# B&R Automation Studio project TD52 (part 10)

```c
/******************************************************************************
 * END OF CODE
 ******************************************************************************/
/*
Local Variables:
c-file-style: bsd
c-basic-offset: 2
comment-column: 45
End:
 */
```

#### MBTMaster.h
```c
/*****************************************************************************
 * Copyright:    B&R Industrie-Automation AG
 *
 * Project:      Library MBTCP
 *
 * Target:       B&R-PCC
 *
 * AR-Version:   B 2.01
 *
 * AS-Version:   V 3.0.71.16.SP01
 *
 * Filename:     MBTMaster.h
 *
 * Function:     module-description
 *
 * Dependencies: description of all dependencies
 *
 *****************************************************************************
 * History:
 *
 * Version | Date        | Author      | Description
 * --------------------------------------------------------------------------
 *    1.00 | 2008-Sep-30 | H.Anderes    | creation
 *****************************************************************************/

/*****************************************************************************
 * includes
 *****************************************************************************/
#ifndef MBTMASTER_H_
#define MBTMASTER_H_
/* ansi-c import */
#include <string.h>
/* system import */
#include <bur/plc.h>                         /* IEC data types */
#include <asstring.h>
#include <brsystem.h>
#include <astcp.h>
#include <convert.h>
#include <sys_lib.h>
/* user defined import */
#include "MBTCP.h"

/*#define _MBTCP_LOGGER_DEBUG*/    /* if defined, errors are logged into the logger */
/*#define _MBTCP_LOGGER_EVENT*/    /* if defined, events are logged into the logger */

#ifdef __i386__
#define SWAPUINT        swapUINT
#define SWAPINT         swapINT
#else
#define SWAPUINT
#define SWAPINT
#endif

/*****************************************************************************
 * constants / macros
 *****************************************************************************/
#define NELEMS(array)           (sizeof(array) / sizeof(array[0]))
/* Booleans, switches
 */
enum {
  FALSE                   = 0,
  TRUE                    = 1,
  EXIT_FAILURE            = 1,
  ON                      = 0xFF00,
  OFF                     = 0x0000
};

#define MAX_COILS    2000
#define MAX_REGISTER 127
/*****************************************************************************
 * type definitions
 *****************************************************************************/
/* STEP values
 */
enum {
  INIT                    = 0,
  WAIT_SERVER             = 5,
  OPEN_PORT               = 10,
  IOCTL                   = 15,
  WAIT_CONNECTION         = 20,
  WAIT_REQUEST            = 30,
  SEND_ANSWER             = 40,
  SEND_REQUEST            = 50,
  WAIT_ANSWER             = 60,
  CLOSE_PORT              = 70,
  FATAL_ERROR0            = 240,
  FATAL_ERROR1            = 241,
  FATAL_ERROR2            = 242,
  FATAL_ERROR3            = 243,
  FATAL_ERROR4            = 244,
  FATAL_ERROR5            = 245,
  FATAL_ERROR6            = 246,
  FATAL_ERROR7            = 247,
  FATAL_ERROR8            = 248,
  FATAL_ERROR9            = 249,
  FATAL_ERROR10           = 250,
  FATAL_ERROR             = 251,
  FINAL_ERROR			  = 252,

  DISABLE                 = 65534,
  BUSY                    = 65535
};

/* Modbus function codes
 */
enum {
  READ_COILS                            = 0x01,
  READ_DISCRETE_INPUTS                  = 0x02,
  READ_HOLDING_REGISTERS                = 0x03,
  READ_INPUT_REGISTERS                  = 0x04,
  WRITE_SINGLE_COIL                     = 0x05,
  WRITE_SINGLE_REGISTER                 = 0x06,
  WRITE_MULTIPLE_COILS                  = 0x0F,
  WRITE_MULTIPLE_REGISTERS              = 0x10,
  READ_WRITE_MULTIPLE_REGISTERS         = 0x17
};
/* Modbus protocol exception codes
 */
enum {
  MB_ILLEGAL_FUNCTION                   = 0x01,
  MB_ILLEGAL_DATA_ADDRESS               = 0x02,
  MB_ILLEGAL_DATA_VALUE                 = 0x03,
  MB_SLAVE_DEVICE_FAILURE               = 0x04,
  MB_ACKNOWLEDGE                        = 0x05,
  MB_SLAVE_DEVICE_BUSY                  = 0x06,
  MB_MEMORY_PARITY_ERROR                = 0x08,
  MB_GATEWAY_PATH_UNAVAILABLE           = 0x0A,
  MB_GATEWAY_TARGET_DEV_FAILED_RESPOND  = 0x0B
};
/* Dimensions
 */
enum {
  MBT_SLAVE_PORT        = 502,
  MAX_OPEN_RETRIES      = 3,
  RECV_TIMEOUT_DFLT     = 500,               /* default timeout */
  IPADDR_L              = 18,
  MAX_NBR_REQUESTS      = 5,                 /* was 20 */
  MAX_BUFFER_LEN        = 1200,/*128,*/
  MESS_LEN              = 100,               /* error message length */
};

/* Datatypes */
typedef struct MBTMasterActionParam_typ
{
  USINT usiFCode;
  USINT usiUnit;
  UINT  uiReadAddr;
  UINT  uiReadQty;
  UDINT puiReadVal;
  UINT  uiWriteAddr;
  UINT  uiWriteQty;
  UDINT puiWriteVal;
  UDINT udiTimer;
} MBTMasterActionParam_typ;

typedef struct MBTMasterActionEnable_typ
{
  BOOL bCyclic;
  BOOL bSingle;
} MBTMasterActionEnable_typ;

typedef struct tstMBT_MData
{
  MBTMasterActionEnable_typ actEnable[MAX_NBR_REQUESTS];
  MBTMasterActionParam_typ actParam[MAX_NBR_REQUESTS];
} tstMBT_MData;

typedef struct
{
  BOOL                  bEnable;
  STRING                slvIPAddr[IPADDR_L];
  UINT                  uiPort;
  UINT                  uiRecvTimeout;
  UDINT                 udiCycleTime;
  tstMBT_MData*         pData;
  UINT                  uiStep;
  TcpOpen_typ           stTcpOpen;
  TcpIoctl_typ          stTcpIoctl;
  TcpClient_typ         stTcpClient;
  TcpSend_typ           stTcpSend;
  TcpRecv_typ           stTcpRecv;
  TcpClose_typ          stTcpClose;
  USINT                 usiLastReq;
  UDINT                 udiRecvTimer;
  UDINT                 udiSendTimer[MAX_NBR_REQUESTS];
  USINT                 usiSendBuf[MAX_BUFFER_LEN];
  USINT                 usiRecvBuf[MAX_BUFFER_LEN];
  BOOL                  bRecvOK;
  UINT                  uiStatus;
  UINT                  uiTxID;
  UDINT                 udiWrongMsg;
  STRING                szMsg[MESS_LEN];
  tcpLINGER_typ         mLinger;
  USINT                 usiOpenRetries;
  USINT                 usiSendCnt;
} tstMBT_MVars;

/*****************************************************************************
 * functions protoytpes
 ****************************************************************************/
void  fMBTMStates(tstMBT_MVars* inst);
UINT create_request_to_server(tstMBT_MVars*   inst,
                               tstMBT_MData*   config,
                               USINT           usiOp,
                               USINT*          usiSendBuf,
                               UINT            uiTxID);
USINT analyze_answer_from_server(tstMBT_MVars* inst,
                                 tstMBT_MData* config,
                                 USINT         usiOp,
                                 USINT*        usiRecvBuf,
                                 UINT          uiTxID);

/****************************************************************************
 * END OF CODE
 ****************************************************************************/
/*
Local Variables:
c-file-style: bsd
c-basic-offset: 2
comment-column: 45
End:
 */
#endif /* MBTMASTER_H_ */
```

#### MBTMaster.c
```c
/******************************************************************************
 * Copyright:    B&R Industrie-Automation AG
 *
 * Project:      Library MBTCP
 *
 * Target:       B&R-PCC
 *
 * AR-Version:   B 2.01
 *
 * AS-Version:   V 3.0.71.16.SP01
 *
 * Filename:     MBTMaster.c
 *
 * Function:     module-description
 *
 * Dependencies: description of all dependencies
 *
 ******************************************************************************
 * History:
 *
 * Version | Date        | Author      | Description
 * ----------------------------------------------------------------------------
 *    1.00 | 2008-Sep-30 | H.Anderes   | creation
 *    2.00 | 2010-okt-04 | H.Anderes   | refactory
 *    5.00 | 2021-may-07 | W.Froehlich | set correct FUB state fMBTSClose.uiStatus
 *****************************************************************************/

/******************************************************************************
 * includes
 *****************************************************************************/
/* ansi-c import */
/* system import */
/* user defined import */
#include "MBTMaster.h"

/******************************************************************************
 * functions
 ******************************************************************************/
/*============================================================================*/
void fMBTMStates(tstMBT_MVars* inst)
/*----------------------------------------------------------------------------
  Function:

  History:

  Version | Date        | Author      | Description
  ----------------------------------------------------------------------------
  1.00    | 2008-sep-30 | H.Anderes    | creation
  2.00    | 2010-okt-04 | H.Anderes   | refactory
  ============================================================================*/
{
  /* _LOCAL */
  UINT uiFatalErrNum;
  USINT i, usiOp;                            /* usiOp: number of operations */
  USINT recv_status;
  /* _DYNAMIC */
  /*==========================================================================*/
  /* check if a null pointer is passed to the fub */
  if (inst == NULL)
  {
    return;
  }
  /*--------------------------------------------------------------------------------
    state machine : Modbus TCP Master
  ---------------------------------------------------------------------------------*/
  switch(inst->uiStep)
  {
  /*-----------------------------------------------------------------------------
    INIT: initialize TcpSend and TCPRecv
  ------------------------------------------------------------------------------*/
  case INIT:
    inst->stTcpSend.pData   = (UDINT)inst->usiSendBuf;
    inst->stTcpRecv.pData   = (UDINT)inst->usiRecvBuf;
    inst->stTcpRecv.datamax = MAX_BUFFER_LEN;
    inst->uiStep            = DISABLE;
    /* FALL THROUGH */
  /*-----------------------------------------------------------------------------
    DISBALE: waits until the fub is enabled
  ------------------------------------------------------------------------------*/
  case DISABLE:
    if(inst->bEnable)
    {
      inst->uiStep = OPEN_PORT;
    }
    break;
  /*-----------------------------------------------------------------------------
    OPEN: opens a TCP - socket
  ------------------------------------------------------------------------------*/
  case OPEN_PORT:
    inst->stTcpOpen.enable = 1;
    inst->stTcpOpen.port   = 0;
    /* call TcpOpen() */
    TcpOpen(&inst->stTcpOpen);
    /* verfiy status */
    switch (inst->stTcpOpen.status)
    {
    /*-------------------------------------------------------------------------*/
    case ERR_OK:
      inst->stTcpClient.enable     = 1;
      inst->stTcpClient.ident      = inst->stTcpOpen.ident;
      inst->stTcpClient.pServer    = (UDINT)inst->slvIPAddr;
      inst->stTcpClient.portserv   = inst->uiPort;
      inst->stTcpSend.ident        = inst->stTcpOpen.ident;
      inst->stTcpRecv.ident        = inst->stTcpOpen.ident;
      inst->uiStep                 = IOCTL;
      /************************************************************************/
      #ifdef _MBTCP_LOGGER_EVENT
	     ERRxwarning( mbtEVENT_OPEN_PORT,
                   inst->stTcpOpen.ident,
                   "MBTCP Client: Open Port");
      #endif
      /************************************************************************/
      break;
    /*-------------------------------------------------------------------------*/
    case ERR_FUB_BUSY:
      /* do nothing */
      break;
    /*-------------------------------------------------------------------------*/
    case tcpERR_NOMORE_IDENTS:
    case tcpERR_ALREADY_EXIST:
    case tcpERR_SOCKET_CREATE:
    case tcpERR_SOCKET_BIND:
    case tcpERR_INTERFACE:
    case tcpERR_SYSTEM:
    case ERR_FUB_ENABLE_FALSE:
    default:
      inst->uiStatus = inst->stTcpOpen.status;
      inst->uiStep   = FATAL_ERROR0;
      break;
    }
    break;
  /*-----------------------------------------------------------------------------
    IOCTRL: configuration of the TCP - connection
  ------------------------------------------------------------------------------*/
  case IOCTL:
    /* set linger that the connection is not abort immediately */
    inst->mLinger.lOnOff     = 0;
    inst->mLinger.lLinger    = 0;
     /* initialize fub */
    inst->stTcpIoctl.enable 	= 1;
    inst->stTcpIoctl.ident	  = inst->stTcpOpen.ident;
    inst->stTcpIoctl.ioctl 	 = tcpSO_LINGER_SET;
    inst->stTcpIoctl.pData	  = (UDINT)&inst->mLinger;
    inst->stTcpIoctl.datalen	= sizeof(tcpLINGER_typ);
    /* call  TcpIoctl()n */
    TcpIoctl(&inst->stTcpIoctl);
    /* verify status */
    switch (inst->stTcpIoctl.status)
    {
    /*-------------------------------------------------------------------------*/
    case ERR_OK:
      inst->usiOpenRetries = 0;      /* we reset prior to next step */
      inst->uiStep         = WAIT_CONNECTION;
      break;
    /*-------------------------------------------------------------------------*/
    case ERR_FUB_BUSY:
      inst->uiStep = IOCTL;
      break;
    /*-------------------------------------------------------------------------*/
    case tcpERR_INVALID_IDENT:
      inst->uiStatus = inst->stTcpIoctl.status;
      if (inst->usiOpenRetries < MAX_OPEN_RETRIES)
      {
        inst->uiStep = OPEN_PORT;
        inst->usiOpenRetries++;
        /************************************************************************/
        #ifdef _MBTCP_LOGGER_DEBUG
		      ERRxwarning( mbtERR_OPEN_RETRIES_IOC,
                     inst->stTcpOpen.ident,
                     "MBTCP Client: OPEN Retries IOCTL");
        #endif
        /************************************************************************/
      }
      else
      {
        inst->uiStep = FATAL_ERROR1;
      }
      break;
    /*-------------------------------------------------------------------------*/
    case tcpERR_PARAMETER:
      inst->uiStatus = inst->stTcpIoctl.status;
      inst->uiStep   = CLOSE_PORT;
      break;
    /*-------------------------------------------------------------------------*/
    case tcpERR_INVALID_IOCTL:
    case ERR_FUB_ENABLE_FALSE:
    default:
      inst->uiStatus = inst->stTcpIoctl.status;
      inst->uiStep   = FATAL_ERROR2;
      break;
    }
    break;
  /*-----------------------------------------------------------------------------
    WAIT: waits until a connection to a TCP Server is acc
  ------------------------------------------------------------------------------*/
  case WAIT_CONNECTION:
    inst->stTcpClient.enable = 1;
    /* call TcpClient() */
    TcpClient(&inst->stTcpClient);
    /* verify status */
    switch (inst->stTcpClient.status)
    {
    /*-------------------------------------------------------------------------*/
    case ERR_OK:
      inst->uiStep = SEND_REQUEST;
      break;
    /*-------------------------------------------------------------------------*/
    case ERR_FUB_BUSY:
      /* do nothing */
	     strcpy( inst->szMsg,
              "WAIT_CONNECTION:TcpClient: Wait Connection");
      break;
    /*-------------------------------------------------------------------------*/
    case tcpERR_INVALID:
   	  inst->uiStep = CLOSE_PORT;
      /*************************************************************************/
      #ifdef _MBTCP_LOGGER_DEBUG
   	  ERRxwarning( tcpERR_INVALID,
                   inst->stTcpClient.ident,
                   "MBTCP Client: Wait connecction; Invalid ");
      #endif
      /*************************************************************************/
      break;
    /*-------------------------------------------------------------------------*/
    case tcpERR_ALREADY_CONNECTED:
      inst->uiStep = CLOSE_PORT;
      /*************************************************************************/
      #ifdef _MBTCP_LOGGER_DEBUG
	     ERRxwarning( tcpERR_ALREADY_CONNECTED,
                             inst->stTcpClient.ident,
                             "MBTCP Client: Wait connecction; Already connected");
      #endif
      /*************************************************************************/
      break;
    /*-------------------------------------------------------------------------*/
    case tcpERR_SYSTEM:
    case ERR_FUB_ENABLE_FALSE:
    default:
      inst->uiStep = FATAL_ERROR3;
      break;
    }
    break;
  /*-----------------------------------------------------------------------------
    CREATE: creates the request
  ------------------------------------------------------------------------------*/
  case SEND_REQUEST:
    if (inst->bEnable)
    {
      inst->bRecvOK = FALSE;
      /* cycle through list of Modbus operations for MAX_NBR_REQUESTS times */
      for (i = inst->usiLastReq + 1;
           i < (MAX_NBR_REQUESTS + inst->usiLastReq + 1);
           i++)
      {
        usiOp = i % MAX_NBR_REQUESTS;
        if ((*(inst->pData)).actEnable[usiOp].bSingle)
        {
          inst->udiSendTimer[usiOp] =
            (*(inst->pData)).actParam[usiOp].udiTimer;
        }
        if ( (((*(inst->pData)).actEnable[usiOp].bCyclic)
              || ((*(inst->pData)).actEnable[usiOp].bSingle)))
        {
          if (inst->udiSendTimer[usiOp]
              >= (*(inst->pData)).actParam[usiOp].udiTimer)
          {
            inst->usiLastReq = usiOp;
            inst->uiStep = SEND_REQUEST + 1;
            inst->uiTxID++;
            inst->stTcpSend.datalen =
                create_request_to_server((tstMBT_MVars*)(inst),
                                       (tstMBT_MData*)(inst->pData),
                                       usiOp,
                                       inst->usiSendBuf,
                                       inst->uiTxID);
            inst->udiSendTimer[usiOp] = 0;
            break;
          }
          else
          {
            inst->udiSendTimer[usiOp] += inst->udiCycleTime;
          }
        }
        else
        {
          inst->udiSendTimer[usiOp]
            = (*(inst->pData)).actParam[usiOp].udiTimer;
        }
      }
    }
    else
    {
      inst->uiStep = CLOSE_PORT;
    }
    break;
  /*-----------------------------------------------------------------------------
    SEND: sends the created request to the server/slave
  ------------------------------------------------------------------------------*/
  case SEND_REQUEST + 1:
    if (inst->bEnable)
    {
      inst->stTcpSend.enable = 1;
      /* call TcpSend() */
      TcpSend(&inst->stTcpSend);
      /* verfiy status */
      switch (inst->stTcpSend.status)
      {
      /*-------------------------------------------------------------------------*/
      case ERR_OK:
        inst->usiSendCnt   = 0;
        inst->udiRecvTimer = 0;
        inst->uiStep       = WAIT_ANSWER;
        break;
      /*-------------------------------------------------------------------------*/
      case ERR_FUB_BUSY:
	       /* do nothing */
		      strcpy( inst->szMsg,
                "SEND_REQUEST + 1:TcpSend: ERR_FUB_BUSY");
	  	    break;
      /*-------------------------------------------------------------------------*/
      case tcpERR_WOULDBLOCK:
         /* send again */
         /************************************************************************/
         #ifdef _MBTCP_LOGGER_DEBUG
  	      ERRxwarning( tcpERR_WOULDBLOCK,
                      inst->stTcpClient.ident,
                      "MBTCP Client: Wouldblock");
         #endif
         /***********************************************************************/
   	   	break;
      /*-------------------------------------------------------------------------*/
      case tcpERR_SENTLEN:
        /* send length not ok. send again */
        /************************************************************************/
        #ifdef _MBTCP_LOGGER_DEBUG
        ERRxwarning( tcpERR_SENTLEN,
                     inst->stTcpClient.ident,
                     "MBTCP Client: Send lenght not Ok");
        #endif
        /************************************************************************/
        break;
      /*------------------------------------------------------------------------*/
      case tcpERR_NOT_CONNECTED:
        inst->uiStep = CLOSE_PORT;
        /************************************************************************/
        #ifdef _MBTCP_LOGGER_DEBUG
		      ERRxwarning( tcpERR_NOT_CONNECTED,
                     inst->stTcpClient.ident,
                     "MBTCP Client: Not connected");
        #endif
        /************************************************************************/
        break;
      /*-------------------------------------------------------------------------*/
      case tcpERR_INVALID_IDENT:
      case tcpERR_PARAMETER:
      case tcpERR_SYSTEM:
      default:
        inst->uiStep = FATAL_ERROR4;
        break;
      }
    }
    else
    {
      inst->uiStep = CLOSE_PORT;
    }
    break;
  /*-----------------------------------------------------------------------------
    WAIT: waits until a response is received or a timeout occured
  ------------------------------------------------------------------------------*/
  case WAIT_ANSWER:
    if (inst->bEnable)
    {
      inst->udiRecvTimer += inst->udiCycleTime;
      if (inst->udiRecvTimer >= inst->uiRecvTimeout)
      {
        /* send again after timeout */
        inst->uiStep = SEND_REQUEST;
        /************************************************************************/
        #ifdef _MBTCP_LOGGER_DEBUG
		      ERRxwarning( mbtERR_TIMEOUT,
                     inst->stTcpClient.ident,
                     "MBTCP Client: Receive Timeout");
        #endif
        /************************************************************************/
        break;
      }
      inst->stTcpRecv.enable = 1;
      /* call TcpRecv() */
      TcpRecv(&(inst->stTcpRecv));
      /* verfiy status */
      switch (inst->stTcpRecv.status)
      {
      /*-------------------------------------------------------------------------*/
      case ERR_OK:
        if (inst->stTcpRecv.recvlen > 8)
        {
          recv_status =
            analyze_answer_from_server((tstMBT_MVars*)(inst),
                                       (tstMBT_MData*)(inst->pData),
                                       inst->usiLastReq,
                                       inst->usiRecvBuf,
                                       inst->uiTxID);
        }
        else
        {
          recv_status = 1;
        }
        if(recv_status)
		      {
           inst->udiWrongMsg++;
           /**********************************************************************/
           #ifdef _MBTCP_LOGGER_DEBUG
 		        ERRxwarning( mbtERR_RESPONSE,
                        inst->stTcpRecv.ident,
                        "MBTCP Client: Response not Ok");
           #endif
           /**********************************************************************/

        }
        else
        {
          (*(inst->pData)).actEnable[inst->usiLastReq].bSingle = 0;
        }
        inst->uiStep = SEND_REQUEST;
        break;
      /*-------------------------------------------------------------------------*/
      case ERR_FUB_BUSY:
      case ERR_FUB_ENABLE_FALSE:
      case tcpERR_NO_DATA:
        /* do nothing */
		      strcpy(inst->szMsg, "WAIT_ANSWER:TcpClient: tcpERR_NO_DATA");
        break;
      /*-------------------------------------------------------------------------*/
      case tcpERR_NOT_CONNECTED:
        inst->uiStep = SEND_REQUEST;
		      strcpy(inst->szMsg, "WAIT_ANSWER:TcpClient: tcpERR_NOT_CONNECTED");
        break;
      /*-------------------------------------------------------------------------*/
      case tcpERR_INVALID_IDENT:
      case tcpERR_PARAMETER:
      case tcpERR_INVALID:
      case tcpERR_NO_OOBDATA:
      case tcpERR_SYSTEM:
      default:
        inst->uiStep = FATAL_ERROR5;
        break;
      }
    }
    else
    {
      inst->uiStep = CLOSE_PORT;
    }
    break;
  /*-----------------------------------------------------------------------------
    CLOSE: closes the TCP - Socket
  ------------------------------------------------------------------------------*/
  case CLOSE_PORT:
    inst->stTcpClose.enable = 1;
    inst->stTcpClose.ident  = inst->stTcpOpen.ident;
    /*
      inst->stTcpClose.how    = tcpSHUT_RD | tcpSHUT_WR;
    */
    inst->stTcpClose.how    = 0;
    /* call TcpClose() */
    TcpClose(&inst->stTcpClose);
    /* verfiy status */
    switch (inst->stTcpClose.status)
    {
    /*-------------------------------------------------------------------------*/
    case ERR_OK:
      inst->uiStep = DISABLE;
      /*************************************************************************/
      #ifdef _MBTCP_LOGGER_DEBUG
	     ERRxwarning( mbtEVENT_CLOSE_PORT,
                   inst->stTcpClose.ident,
                   "MBTCP Client: Close Port");
      #endif
      /*************************************************************************/
      break;
    /*-------------------------------------------------------------------------*/
    case ERR_FUB_BUSY:
      /* do nothing */
      break;
    /*-------------------------------------------------------------------------*/
    case tcpERR_INVALID_IDENT:
      inst->uiStep = WAIT_CONNECTION;
      break;
    /*-------------------------------------------------------------------------*/
    case ERR_FUB_ENABLE_FALSE:
    default:
      inst->uiStep = FATAL_ERROR6;
      break;
    }
    break;
  /*-----------------------------------------------------------------------------
    FATAL ERROR: a fatal error occured
  ------------------------------------------------------------------------------*/
  case FATAL_ERROR0:
  case FATAL_ERROR1:
  case FATAL_ERROR2:
  case FATAL_ERROR3:
  case FATAL_ERROR4:
  case FATAL_ERROR5:
  case FATAL_ERROR6:
  default:
   /* vefiy in which state the fatal error occured */
  	switch(inst->uiStep)
	  {
	  case FATAL_ERROR0: uiFatalErrNum = 0; break;
  	case FATAL_ERROR1: uiFatalErrNum = 1; break;
  	case FATAL_ERROR2: uiFatalErrNum = 2; break;
  	case FATAL_ERROR3: uiFatalErrNum = 3; break;
  	case FATAL_ERROR4: uiFatalErrNum = 4; break;
  	case FATAL_ERROR5: uiFatalErrNum = 5; break;
  	case FATAL_ERROR6: uiFatalErrNum = 6; break;
	  default:
		   uiFatalErrNum = 7; break;
	  }
	   /*************************************************************************/
    #ifdef _MBTCP_LOGGER_DEBUG
   	ERRxwarning( mbtERR_FATAL_ERROR,
                 uiFatalErrNum,
                 "MBTCP Client: FATAL ERROR State Machine");
    #endif
    /*************************************************************************/
   	inst->uiStep = FINAL_ERROR;
    break;

  case FINAL_ERROR:
  	/*Do nothing until Reboot RPS*/
  	break;
  }
}

/*============================================================================*/
UINT create_request_to_server(tstMBT_MVars* inst,
                               tstMBT_MData* config,
                               USINT         usiOp,
                               USINT*        usiSendBuf,
                               UINT          uiTxID)
/*----------------------------------------------------------------------------
  Function:

  History:

  Version | Date        | Author      | Description
  ----------------------------------------------------------------------------
     1.00 | 2008-sep-30 | H.Anderes    | creation
  ============================================================================*/
{
  UINT  uint_var, data_len, i;
  INT  int_var;
  UINT  value;
  UINT  val;
 /*==========================================================================*/
  data_len = 0;

  memset(usiSendBuf, 0, MAX_BUFFER_LEN);
  /* Transaction id: 2 bytes */
  uint_var = SWAPUINT(uiTxID);
  memmove(&usiSendBuf[0], &uint_var, sizeof(uint_var));
  /* Protocol id: 2 bytes */
  uint_var = 0;
  memmove(&usiSendBuf[2], &uint_var, sizeof(uint_var));
  /* Length: 2 bytes */
  /* Unit: 1 byte */
  usiSendBuf[6] = (*config).actParam[usiOp].usiUnit;

  switch((*config).actParam[usiOp].usiFCode)
  {
  /*-------------------------------------------------------------------------
      READ: read coils
  --------------------------------------------------------------------------*/
  case READ_COILS:
    /* Function code: 1 byte */
    usiSendBuf[7] = READ_COILS;
    /* Starting address: 2 bytes */
    uint_var = SWAPUINT((*config).actParam[usiOp].uiReadAddr);
    memmove(&usiSendBuf[8], &uint_var, sizeof(uint_var));
    /* Coils number: 2 bytes */
    uint_var = SWAPUINT((*config).actParam[usiOp].uiReadQty);
    memmove(&usiSendBuf[10], &uint_var, sizeof(uint_var));
    /* Data len */
    data_len = 6;
    inst->bRecvOK = FALSE;
    break;
  /*-------------------------------------------------------------------------
      READ: read discrete inputs
  --------------------------------------------------------------------------*/
  case READ_DISCRETE_INPUTS:
    /* Function code: 1 byte */
    usiSendBuf[7] = READ_DISCRETE_INPUTS;
    /* Starting address: 2 bytes */
    uint_var = SWAPUINT((*config).actParam[usiOp].uiReadAddr);
    memmove(&usiSendBuf[8], &uint_var, sizeof(uint_var));
    /* Inputs number: 2 bytes */
    uint_var = SWAPUINT((*config).actParam[usiOp].uiReadQty);
    memmove(&usiSendBuf[10], &uint_var, sizeof(uint_var));
    /* Data len */
    data_len = 6;
    inst->bRecvOK = FALSE;
    break;
  /*-------------------------------------------------------------------------
      READ: read holding registers
  --------------------------------------------------------------------------*/
  case READ_HOLDING_REGISTERS:
    /* Function code: 1 byte */
    usiSendBuf[7] = READ_HOLDING_REGISTERS;
    /* Starting address: 2 bytes */
    uint_var = SWAPUINT((*config).actParam[usiOp].uiReadAddr);
    memmove(&usiSendBuf[8], &uint_var, sizeof(uint_var));
    /* Holding registers number: 2 bytes */
    uint_var = SWAPUINT((*config).actParam[usiOp].uiReadQty);
    memmove(&usiSendBuf[10], &uint_var, sizeof(uint_var));
    /* Data len */
    data_len = 6;
    inst->bRecvOK = FALSE;
    break;
  /*-------------------------------------------------------------------------
      READ: read input registers
  --------------------------------------------------------------------------*/
  case READ_INPUT_REGISTERS:
    /* Function code: 1 byte */
    usiSendBuf[7] = READ_INPUT_REGISTERS;
    /* Starting address: 2 bytes */
    uint_var = SWAPUINT((*config).actParam[usiOp].uiReadAddr);
    memmove(&usiSendBuf[8], &uint_var, sizeof(uint_var));
    /* Input registers number: 2 bytes */
    uint_var = SWAPUINT((*config).actParam[usiOp].uiReadQty);
    memmove(&usiSendBuf[10], &uint_var, sizeof(uint_var));
    /* Data len */
    data_len = 6;
    inst->bRecvOK = FALSE;
    break;
  /*-------------------------------------------------------------------------
      WRITE: write single coil
  --------------------------------------------------------------------------*/
  case WRITE_SINGLE_COIL:
    /* Function code: 1 byte */
    usiSendBuf[7] = WRITE_SINGLE_COIL;
    /* Starting address: 2 bytes */
    uint_var = SWAPUINT((*config).actParam[usiOp].uiWriteAddr);
    memmove(&usiSendBuf[8], &uint_var, sizeof(uint_var));
    /* Value: 2 bytes */
    memmove(&val, (UINT *)((*config).actParam[usiOp].puiWriteVal), sizeof(UINT));
    if ((BOOL)(val))
      value = ON;
    else
      value = OFF;
    int_var = SWAPUINT(value);
    memmove(&usiSendBuf[10], &int_var, sizeof(int_var));
    /* Data len */
    data_len = 6;
    inst->bRecvOK = FALSE;
    break;
  /*-------------------------------------------------------------------------
      WRITE: write single register
  --------------------------------------------------------------------------*/
  case WRITE_SINGLE_REGISTER:
    /* Function code: 1 byte */
    usiSendBuf[7] = WRITE_SINGLE_REGISTER;
    /* Starting address: 2 bytes */
    uint_var = SWAPUINT((*config).actParam[usiOp].uiWriteAddr);
    memmove(&usiSendBuf[8], &uint_var, sizeof(uint_var));
    /* Value: 2 bytes */
    memmove(&val, (UINT *)(*config).actParam[usiOp].puiWriteVal, sizeof(UINT));
    value = (UINT)(val);
    uint_var = SWAPUINT(value);
    memmove(&usiSendBuf[10], &uint_var, sizeof(uint_var));
    /* Data len */
    data_len = 6;
    inst->bRecvOK = FALSE;
    break;
  /*-------------------------------------------------------------------------
      WRITE: write multiple coils
  --------------------------------------------------------------------------*/
  case WRITE_MULTIPLE_COILS:
    /* Function code: 1 byte */
    usiSendBuf[7] = WRITE_MULTIPLE_COILS;
    /* Starting address: 2 bytes */
    uint_var = SWAPUINT((*config).actParam[usiOp].uiWriteAddr);
    memmove(&usiSendBuf[8], &uint_var, sizeof(uint_var));
    /* Quantity: 2 bytes */
    uint_var = SWAPUINT((*config).actParam[usiOp].uiWriteQty);
    memmove(&usiSendBuf[10], &uint_var, sizeof(uint_var));
    /* Byte count: 1 byte */
    /* Number of usiSendBuf bytes needed to contain data */
    /* less than 8 binary digits: 1 byte */
    if ( (*config).actParam[usiOp].uiWriteQty % 8)
      usiSendBuf[12] = ((*config).actParam[usiOp].uiWriteQty / 8) + 1;
    else      /* more than 8 binary digits: quantity / 8 bytes */
      usiSendBuf[12] = (*config).actParam[usiOp].uiWriteQty / 8;
    /* Coil value: x byte */
    for (i = 0; i < (*config).actParam[usiOp].uiWriteQty; i++)
    {
      memmove(&val,
              (UINT *)((*config).actParam[usiOp].puiWriteVal  +  i * sizeof(UINT)),
              sizeof(UINT));
      if ((BOOL)(val))
        usiSendBuf[13 + (i/8)]
          = usiSendBuf[13 + (i/8)] | (USINT)(0x01 << (i%8));
      else
        usiSendBuf[13 + (i/8)]
          = usiSendBuf[13 + (i/8)] & (USINT)~(0x01 << (i%8));
    }
    /* Data len */
    data_len = 7 + usiSendBuf[12];
    inst->bRecvOK = FALSE;
    break;
  /*-------------------------------------------------------------------------
      WRITE: write multiple registers
  --------------------------------------------------------------------------*/
  case WRITE_MULTIPLE_REGISTERS:
    /* Function code: 1 byte */
    usiSendBuf[7] = WRITE_MULTIPLE_REGISTERS;
    /* Starting address: 2 bytes */
    uint_var = SWAPUINT((*config).actParam[usiOp].uiWriteAddr);
    memmove(&usiSendBuf[8], &uint_var, sizeof(uint_var));
    /* Quantity: 2 bytes */
    uint_var = SWAPUINT((*config).actParam[usiOp].uiWriteQty);
    memmove(&usiSendBuf[10], &uint_var, sizeof(uint_var));
    /* Byte count: 1 byte */
    usiSendBuf[12] = (*config).actParam[usiOp].uiWriteQty * 2;
    /* Coil value: x byte */
    for(i = 0; i < (*config).actParam[usiOp].uiWriteQty; i++)
    {
      value = ((INT*)((*config).actParam[usiOp].puiWriteVal))[i];
      int_var = SWAPINT(value);
      memmove(&usiSendBuf[13 + (i*2)], &int_var, sizeof(int_var));
    }
    /* Data len */
    data_len = 7 + usiSendBuf[12];
    inst->bRecvOK = FALSE;
    break;
  /*-------------------------------------------------------------------------
     READ WRITE:read  write multiple registers
  --------------------------------------------------------------------------*/
  case READ_WRITE_MULTIPLE_REGISTERS:
    /* Function code: 1 byte */
    usiSendBuf[7] = READ_WRITE_MULTIPLE_REGISTERS;
    /* Read starting address: 2 bytes */
    uint_var = SWAPUINT((*config).actParam[usiOp].uiReadAddr);
    memmove(&usiSendBuf[8], &uint_var, sizeof(uint_var));
    /* Read quantity: 2 bytes */
    uint_var = SWAPUINT((*config).actParam[usiOp].uiReadQty);
    memmove(&usiSendBuf[10], &uint_var, sizeof(uint_var));
    /* Write starting address: 2 bytes */
    uint_var = SWAPUINT((*config).actParam[usiOp].uiWriteAddr);
    memmove(&usiSendBuf[12], &uint_var, sizeof(uint_var));
    /* write quantity: 2 bytes */
    uint_var = SWAPUINT((*config).actParam[usiOp].uiWriteQty);
    memmove(&usiSendBuf[14], &uint_var, sizeof(uint_var));
    /* Byte count: 1 byte */
    usiSendBuf[16] = (*config).actParam[usiOp].uiWriteQty * 2;
    /* Coil value: x byte */
    for(i = 0; i < (*config).actParam[usiOp].uiWriteQty; i++)
    {
      value = ((INT*)((*config).actParam[usiOp].puiWriteVal))[i];
      int_var = SWAPINT(value);
      memmove(&usiSendBuf[17 + (i*2)], &int_var, sizeof(int_var));
    }
    /* Data len */
    data_len = 11 + usiSendBuf[16];
    inst->bRecvOK = FALSE;
    break;
  default:
    break;
  }
  /* Length: 2 bytes */
  uint_var = SWAPUINT(data_len);
  memmove(&usiSendBuf[4], &uint_var, sizeof(uint_var));

  return (6 + data_len);
}

 /*==========================================================================*/
USINT analyze_answer_from_server(tstMBT_MVars* inst,
                                 tstMBT_MData* config,
                                 USINT         usiOp,
                                 USINT*        usiRecvBuf,
                                 UINT          uiTxID)
/*----------------------------------------------------------------------------
  Function:

  History:

  Version | Date        | Author      | Description
  ----------------------------------------------------------------------------
     1.00 | 2008-sep-30 | H.Anderes   | creation
     2.00 | 2010-okt-04 | H.Anderes   | refactory
  ============================================================================*/
{
  INT   int_var;
  UINT  uint_var, recv_tr_id, protocol_id, length, uiQty,i;
  USINT unit, function_code;
  UINT  coil_val, di_val;         /* was UDINT */
  /*==========================================================================*/

  coil_val = 0;
  di_val   = 0;
  /* (byte 0,1)  transition is */
  memmove(&uint_var, &(usiRecvBuf[0]), sizeof(uint_var));
  recv_tr_id = SWAPUINT(uint_var);
  /* (byte 2,3)  protocol id */
  memmove(&uint_var, &(usiRecvBuf[2]), sizeof(uint_var));
  protocol_id = SWAPUINT(uint_var);
  /* (byte 4,5)  length */
  memmove(&uint_var, &(usiRecvBuf[4]), sizeof(uint_var));
  length = SWAPUINT(uint_var);
  /* (byte 4,5)  length */
  unit = usiRecvBuf[6];
  /* (byte 7 ) function code */
  function_code = usiRecvBuf[7];

  if (    (recv_tr_id == uiTxID)
       && (protocol_id == 0)
       && (length > 0)
       && (function_code  < 0x80) )
  {

    switch(function_code)
    {
    /*-------------------------------------------------------------------------
      READ: read coils
    --------------------------------------------------------------------------*/
    case READ_COILS:
      /* Quantity: 1 byte */
      uiQty = usiRecvBuf[8];
      if (uiQty > MAX_COILS)
      {
        uiQty = MAX_COILS;
      }
      /* Coil value: x bytes */
      /* uiQty is number of bytes received */
      for (i = 0;(i < uiQty*8) && (i < (*config).actParam[usiOp].uiReadQty); i++) {
        coil_val = (UINT)(usiRecvBuf[9 + (i/8)] & (USINT)(0x01 << (i%8)));
        if ((BOOL)(coil_val))
          ((INT*)((*config).actParam[usiOp].puiReadVal))[i] = 1;
        else
          ((INT*)((*config).actParam[usiOp].puiReadVal))[i] = 0;
      }
      inst->bRecvOK = TRUE;
      break;
    /*-------------------------------------------------------------------------
      READ: read discrete inputs
    --------------------------------------------------------------------------*/
    case READ_DISCRETE_INPUTS:
      /* Quantity: 1 byte */
      uiQty = usiRecvBuf[8];
      if (uiQty > MAX_COILS)
      {
        uiQty = MAX_COILS;
      }
      /* Coil value: x byte */
      /* quantity is number of bytes received */
      for(i = 0; (i < uiQty*8) && (i < (*config).actParam[usiOp].uiReadQty); i++) {
        di_val = (UINT)(usiRecvBuf[9 + (i/8)] & (USINT)(0x01 << (i%8)));
         if ((BOOL)(di_val))
           ((INT*)((*config).actParam[usiOp].puiReadVal))[i] = 1;
         else
           ((INT*)((*config).actParam[usiOp].puiReadVal))[i] = 0;
      }
      inst->bRecvOK = TRUE;
      break;
    /*-------------------------------------------------------------------------
      READ: read hoding registers
    --------------------------------------------------------------------------*/
    case READ_HOLDING_REGISTERS:
      /* Quantity: 1 byte */
       uiQty = usiRecvBuf[8] / 2;
       if (uiQty > MAX_REGISTER)
       {
         uiQty = MAX_REGISTER;
       }
      /* Coil value: x byte */
      for(i = 0; i < uiQty; i++) {
        memmove(&int_var, &usiRecvBuf[9 + (i*2)], sizeof(int_var));
        ((INT*)((*config).actParam[usiOp].puiReadVal))[i] = SWAPINT(int_var);
      }
      inst->bRecvOK = TRUE;
      break;
    /*-------------------------------------------------------------------------
      READ: read input registers
    --------------------------------------------------------------------------*/
    case READ_INPUT_REGISTERS:
      /* Quantity: 1 byte */
      uiQty = usiRecvBuf[8] / 2;
      if (uiQty > MAX_REGISTER)
      {
        uiQty = MAX_REGISTER;
      }
      /* Coil value: x byte */
      for(i = 0; i < uiQty; i++) {
        memmove(&int_var, &usiRecvBuf[9 + (i*2)], sizeof(int_var));
        ((INT*)((*config).actParam[usiOp].puiReadVal))[i] = SWAPINT(int_var);
      }
      inst->bRecvOK = TRUE;
      break;
    /*-------------------------------------------------------------------------
      READ: read write multiple registers
    --------------------------------------------------------------------------*/
    case READ_WRITE_MULTIPLE_REGISTERS:
      /* Quantity: 1 byte */
      uiQty = usiRecvBuf[8] / 2;
      if (uiQty > MAX_REGISTER)
      {
        uiQty = MAX_REGISTER;
      }
      /* Coil value: x byte */
      for(i = 0; i < uiQty; i++) {
        memmove(&int_var, &usiRecvBuf[9 + (i*2)], sizeof(int_var));
        ((INT*)((*config).actParam[usiOp].puiReadVal))[i] = SWAPINT(int_var);
      }
      inst->bRecvOK = TRUE;
      break;

    default:
      inst->bRecvOK = TRUE;
      break;
    }
  }
  else
  { /* if (    (recv_tr_id == uiTxID)
            && (protocol_id == 0)
            && (length > 0)
            && (function_code  < 0x80) ) */
    /*************************************************************************/
    #ifdef _MBTCP_LOGGER_DEBUG
    if(protocol_id != 0)
    {
		    ERRxwarning( mbtERR_PROTOCOL_ID,
                   inst->stTcpRecv.ident,
                   "MBTCP Client: Protocol ID != 0");
    }
	   if(length == 0)
    {
		    ERRxwarning( mbtERR_RESPONSE,
                   inst->stTcpRecv.ident,
                   "MBTCP Client: Response lenght == 0");
    }
	   if(function_code  > 0x80)
    {
		    ERRxwarning( mbtERR_RESPONSE,
                    inst->stTcpRecv.ident,
                    "MBTCP Client: function_code  > 0x80");
    }
    #endif
    /*************************************************************************/

    return EXIT_FAILURE;
  }

  return ERR_OK;
}

/******************************************************************************
 * END OF CODE
 ******************************************************************************/
/*
Local Variables:
c-file-style: bsd
c-basic-offset: 2
comment-column: 45
End:
*/
```

#### Convert.c
```c
/******************************************************************************
 * Copyright:    B&R Industrie-Automation AG
 *
 * Project:      Library MBTCP
 *
 * Target:       B&R-PCC
 *
 * Filename:     Convert.c
 *
 * Function:     module-description
 *
 * Dependencies: description of all dependencies
 *
 ******************************************************************************
 * History:
 *
 * Version | Date        | Author       | Description
 * ----------------------------------------------------------------------------
 *    1.00 | 2012-aug-03 | H.Anderes    | creation
 *****************************************************************************/

/*****************************************************************************
 * includes
 *****************************************************************************/
/* ansi-c import */
/* system import */
#include <bur/plctypes.h>
/* user defined import */
#include "Convert.h"

INT swapINT (INT wInputValue)
{
 return (wInputValue << 8) + (USINT)(wInputValue >> 8);
}

UINT swapUINT (UINT wInputValue)
{
 return (wInputValue << 8) + (USINT)(wInputValue >> 8);
}

/*****************************************************************************
 * END OF CODE
 *****************************************************************************/
```

#### Convert.h
```c
/*****************************************************************************
 * Copyright:    B&R Industrie-Automation AG
 *
 * Project:      Library MBTCP
 *
 * Target:       B&R-PCC
 *
 * Filename:     Convert.h
 *
 * Function:     module-description
 *
 * Dependencies: description of all dependencies
 *
 *****************************************************************************
 * History:
 *
 * Version | Date        | Author      | Description
 * --------------------------------------------------------------------------
 *    1.00 | 2008-sep-19 | H.Anderes    | creation
 *****************************************************************************/

/*****************************************************************************
 * includes
 *****************************************************************************/
#ifndef CONVERT_H_
#define CONVERT_H_

#include <bur/plctypes.h>

INT swapINT (INT wInputValue);
UINT swapUINT (UINT wInputValue);

#endif /* CONVERT_H_ */
/*****************************************************************************
 * END OF CODE
 *****************************************************************************/
```

### Library Logical/Libraries/TPSA_lib (IEC, version 4.07.4) - The TPSA library contains general functions like ring buffers, median calculation, counter blocks etc.

#### TPSA_lib.typ - Exported data types
```iecst
(********************************************************************
 * COPYRIGHT -- INNIO Company
 ********************************************************************
 * Library: TCC_intern
 * File: TCC_intern.typ
 * Author: WaldharM
 * Created: September 14, 2010
 ********************************************************************
 * Data types of library TCC_intern
 ********************************************************************)

TYPE
	_tXY_Stat : STRUCT
		tLn_Nom : _tLn;				(* Nominal line *)
		tLn_Set : _tLn;				(* Setpoint line *)
		tWin : _tWin;				(* window size *)
		tWPt : _tPt;				(* working point *)
	END_STRUCT;
	_tLn : STRUCT
		x : ARRAY [0..1] OF REAL;
		y : ARRAY [0..1] OF REAL;
	END_STRUCT;
	_tWin : STRUCT
		x : ARRAY [0..1] OF REAL;
		y : ARRAY [0..1] OF REAL;
	END_STRUCT;
	_tPt : STRUCT
		x : REAL;
		y : REAL;
	END_STRUCT;
	_tLL_Struct: STRUCT
		rPr_P2s_Ref_0kW : ARRAY [0..4] OF REAL;	(* Reference point 0kW (0), Reference for boost pressure [bar] - depending on the gas type *)
		tRef_a : ARRAY [0..4] OF _tLL_Pt_Struct; (* Reference point a   (1) - depending on the gas type *)
		tRef_b : ARRAY [0..4] OF _tLL_Pt_Struct; (* Reference point b   (2) - depending on the gas type *)
		tRef_c : ARRAY [0..4] OF _tLL_Pt_Struct; (* Reference point c   (3) - depending on the gas type *)
	END_STRUCT;
	_tLL_Pt_Struct: STRUCT
		rP_Eng : REAL;			(* Reference for engine power [kW] *)
		rN_Eng : REAL;			(* Reference for engine speed [rpm]  *)
		rPr_P2s : REAL;			(* Reference for boost pressure [bar]  *)
		rT_T2s : REAL;			(* Reference for mixture temperature [°C]  *)
	END_STRUCT;
END_TYPE
```

#### TPSA_lib.fun - Exported functions and function blocks
```iecst
(********************************************************************
 * COPYRIGHT -- INNIO Company
 ********************************************************************
 * Library: TCC_intern
 * File: TCC_intern.fun
 * Author: WaldharM
 * Created: September 14, 2010
 ********************************************************************
 * Functions and function blocks of library TCC_intern
 ********************************************************************)

FUNCTION_BLOCK MAP_REAL18
	VAR_INPUT
		X_PAR : ARRAY[0..18] OF REAL;
		Y_PAR : ARRAY[0..25] OF REAL;
		Z_PAR : ARRAY[0..475] OF REAL;
		x : REAL;
		y : REAL;
		X_NUM : INT;
		Y_NUM : INT;
	END_VAR
	VAR_OUTPUT
		z : REAL;
	END_VAR
	VAR
		index : INT;
		x_index : INT;
		y_index : INT;
		zx_intp1_tmp : REAL;
		zx_intp2_tmp : REAL;
		z1_tmp : REAL;
		z2_tmp : REAL;
		z3_tmp : REAL;
		z4_tmp : REAL;
	END_VAR
END_FUNCTION_BLOCK

FUNCTION_BLOCK MEDIAN24
	VAR_INPUT
		anzahl : USINT;
		in : ARRAY[0..24] OF INT;
	END_VAR
	VAR_OUTPUT
		median : INT;
	END_VAR
	VAR
		i : USINT;
		j : USINT;
		ssDummy : INT;
	END_VAR
END_FUNCTION_BLOCK

FUNCTION_BLOCK RMEDIAN24
	VAR_INPUT
		anzahl : USINT;
		in : ARRAY[0..24] OF REAL;
	END_VAR
	VAR_OUTPUT
		median : REAL;
	END_VAR
	VAR
		i : USINT;
		j : USINT;
		rDummy : REAL;
	END_VAR
END_FUNCTION_BLOCK

FUNCTION_BLOCK RING500_R
	VAR_INPUT
		in : REAL;
		iCnt_Max : INT;
		reset : BOOL;
	END_VAR
	VAR_OUTPUT
		out : REAL;
	END_VAR
	VAR
		iCnt : INT;
		rBuffer : ARRAY[0..500] OF REAL;
	END_VAR
END_FUNCTION_BLOCK

FUNCTION_BLOCK RING1000_R
	VAR_INPUT
		in : REAL;
		iCnt_Max : INT;
		reset : BOOL;
	END_VAR
	VAR_OUTPUT
		out : REAL;
	END_VAR
	VAR
		iCnt : INT;
		rBuffer : ARRAY[0..1000] OF REAL;
	END_VAR
END_FUNCTION_BLOCK

FUNCTION_BLOCK COUNTER50
	VAR_INPUT
		in : BOOL;
		iNum_Max : SINT;
		ti_Max : TIME;
		reset : BOOL;
	END_VAR
	VAR_OUTPUT
		out : BOOL;
	END_VAR
	VAR
		iCmp : SINT;
		iCnt : SINT;
	END_VAR
	VAR CONSTANT
		iCnt_Max : SINT := 50;
	END_VAR
	VAR
		ti : ARRAY[0..50] OF TIME;
		zzEdge00000 : BOOL;
	END_VAR
END_FUNCTION_BLOCK

FUNCTION_BLOCK COUNTER100
	VAR_INPUT
		in : BOOL;
		iNum_Max : SINT;
		ti_Max : TIME;
		reset : BOOL;
	END_VAR
	VAR_OUTPUT
		out : BOOL;
	END_VAR
	VAR
		iCmp : SINT;
		iCnt : SINT;
	END_VAR
	VAR CONSTANT
		iCnt_Max : SINT := 100;
	END_VAR
	VAR
		ti : ARRAY[0..100] OF TIME;
		zzEdge00000 : BOOL;
	END_VAR
END_FUNCTION_BLOCK

FUNCTION_BLOCK PRed (* Power reduction function block *)
	VAR_INPUT
		iAdr_P_Type : UDINT; (* address of actual Load reduction type *)
		iAdr_P_Set : UDINT; (* address of actual normalized load reduction *)
		iAdr_P_Set_Max : UDINT; (* address of all load reductions*)
		rP_Red : REAL; (* normalized load reduction *)
		iType : INT; (* load reduction type *)
		PT : TIME; (* time off delay for Q *)
		bEna : BOOL; (* enable block *)
		bParaSetupOk_2s : BOOL; (* Para setup OK *)
	END_VAR
	VAR_OUTPUT
		Q : BOOL; (* reduction active *)
	END_VAR
	VAR
		rP_Set_Act : REAL;
		iType_Act : INT;
		xTOF : TOF;
		rP_Set_Max : REAL;
	END_VAR
END_FUNCTION_BLOCK
```

#### mapCyclic.st - Cyclic code
```iecst
(*******************************************************************************
	AGGR: MAP_REAL18 characterisitc map - real 18x18 (FUB)

This code is confidential and proprietary to the INNIO Company.
It may not be used in any form, or reproduced in any manner, without the express
written permission of the INNIO Company.
Copyright, INNIO Company, 2019

- limitation of inputs
- detection of according area in x direction
- assignment of the z values for the according area
- linear interpolation in the according area

History:
-------
V1.00	14-12-2010	Graus, 	generated
V1.01	15-02-2011	Graus,	correction to avoid negativ array index
							via max function with zero input

Instructions for use:
-----------------------

- linear interpolation of a characteristic map
- inputs: x, y: REAL
- outputs: z: REAL
- parameters:	X_PAR, Y_PAR: REAL		supporting points
				Z_PAR: REAL				values (order: [x(0)y(0), x(1)y(0),
													... x(1)y(1), x(2)y(1),
													... x(n-1)y(n), x(n)y(n)] )
				X_NUM, Y_NUM: INT		number of supporting points of the axis

- all specified supporting points have to be set strictly monotonic increasing
- no extrapolation outside of the range of the supporting points
- max. size of the map MAP_REAL12 is limited to 12x12
- size of map has to be specified by X_NUM and Y_NUM

Outstandings:
----------------

*******************************************************************************)

FUNCTION_BLOCK MAP_REAL18

	x := LIMIT(X_PAR[0], x, X_PAR[MAX(0, X_NUM - 1)]);		(* limitation of input / avoid extrapolation *)
	y := LIMIT(Y_PAR[0], y, Y_PAR[MAX(0, Y_NUM - 1)]);		(* limitation of input / avoid extrapolation *)

	FOR index := 0 TO X_NUM - 2 DO								(* detection of according area in x direction *)
		IF X_PAR[index] <= x AND x <= X_PAR[index + 1]   THEN	(* according area detected *)
			x_index := index;									(* assign index *)
			EXIT;												(* exit loop if detected *)
		END_IF;
	END_FOR;

	FOR index := 0 TO Y_NUM - 2 DO								(* detection of according area in y direction *)
		IF Y_PAR[index] <= y AND y <= Y_PAR[index + 1]   THEN	(* according area detected *)
			y_index := index;									(* assign index *)
			EXIT;												(* exit loop if detected *)
		END_IF;
	END_FOR;

	z1_tmp := Z_PAR[ X_NUM * y_index + x_index ];				(* assignment of the z values for the according area *)
	z2_tmp := Z_PAR[ X_NUM * y_index + x_index + 1 ];			(* assignment of the z values for the according area *)
	z3_tmp := Z_PAR[ X_NUM * (y_index + 1) + x_index ];			(* assignment of the z values for the according area *)
	z4_tmp := Z_PAR[ X_NUM * (y_index + 1) + x_index + 1 ];		(* assignment of the z values for the according area *)

	(* linear interpolation in the according area *)
	IF (X_PAR[x_index + 1] - X_PAR[x_index]) <> 0 THEN
		zx_intp1_tmp := ( z2_tmp - z1_tmp ) * ( (x - X_PAR[x_index]) / (X_PAR[x_index + 1] - X_PAR[x_index]) ) + z1_tmp;
		zx_intp2_tmp := ( z4_tmp - z3_tmp ) * ( (x - X_PAR[x_index]) / (X_PAR[x_index + 1] - X_PAR[x_index]) ) + z3_tmp;
	ELSE
		zx_intp1_tmp := z1_tmp;
		zx_intp2_tmp := z3_tmp;
	END_IF;
	IF (Y_PAR[y_index + 1] - Y_PAR[y_index]) <> 0 THEN
		z := ( zx_intp2_tmp - zx_intp1_tmp ) * ( (y - Y_PAR[y_index]) / (Y_PAR[y_index + 1] - Y_PAR[y_index]) ) + zx_intp1_tmp;
	ELSE
		z := zx_intp1_tmp;
	END_IF;

END_FUNCTION_BLOCK
```

#### median.st
```iecst
(********************************************************************
 * COPYRIGHT -- INNIO Company
 ********************************************************************
 * Package: TCC_intern
 * File: median.st
 * Author: WaldharM
 * Created: September 14, 2010
 *******************************************************************)

//
FUNCTION_BLOCK MEDIAN24
	anzahl := LIMIT(0,anzahl,24);
	FOR i := 2 TO anzahl DO
		j := i;
		WHILE j >= 2 AND in[j-1] > in[j] DO
			ssDummy := in[j-1];
			in[j-1] := in[j];
			in[j] 	:= ssDummy;
			j := j-1;
		END_WHILE
	END_FOR

	IF INT_TO_BOOL(anzahl MOD 2) THEN	// ungerade
		median := in[(anzahl+1)/2];
	ELSE 					//gerade
		median := (in[anzahl/2] + in[anzahl/2+1])/2;
	END_IF
END_FUNCTION_BLOCK
```

#### ring.st
```iecst
(********************************************************************
 * COPYRIGHT -- INNIO Company
 ********************************************************************
 * Package: TPSA_lib
 * File: ring.st
 * Author: CaksM
 * Created: Okt 22, 2014
 *******************************************************************)

FUNCTION_BLOCK RING500_R

	IF reset THEN
		//setzte alles zurück
		FOR iCnt:=1 TO 500 DO
			rBuffer[iCnt]	:=	0;
		END_FOR
		iCnt	:=	1;
		out		:=	0;
	ELSE
		//für den ersten start:
		iCnt		:=	LIMIT(1, iCnt, 500);

		//limitiere gegen bereichsverletzung
		iCnt_Max	:=	LIMIT(1, iCnt_Max, 500);

		//schreibe in den buffer:
		rBuffer[iCnt]	:=	in;

		//gehe zum ältesten element
		IF iCnt < iCnt_Max THEN
			iCnt 			:=	iCnt + 1;
		ELSE
			iCnt 			:=	1;
		END_IF

		//lese aus den buffer:
		out					:=	rBuffer[iCnt];
	END_IF

END_FUNCTION_BLOCK

FUNCTION_BLOCK RING1000_R

	IF reset THEN
		//setzte alles zurück
		FOR iCnt:=1 TO 1000 DO
			rBuffer[iCnt]	:=	0;
		END_FOR
		iCnt	:=	1;
		out		:=	0;
	ELSE
		//für den ersten start:
		iCnt		:=	LIMIT(1, iCnt, 1000);

		//limitiere gegen bereichsverletzung
		iCnt_Max	:=	LIMIT(1, iCnt_Max, 1000);

		//schreibe in den buffer:
		rBuffer[iCnt]	:=	in;

		//gehe zum ältesten element
		IF iCnt < iCnt_Max THEN
			iCnt 			:=	iCnt + 1;
		ELSE
			iCnt 			:=	1;
		END_IF

		//lese aus den buffer:
		out					:=	rBuffer[iCnt];
	END_IF

END_FUNCTION_BLOCK
```

#### counter.st
```iecst
(********************************************************************
 * COPYRIGHT -- INNIO Company
 ********************************************************************
 * Package: TPSA_lib
 * File: counter.st
 * Author: CaksM
 * Created: Sept 23, 2014
 *******************************************************************)

FUNCTION_BLOCK COUNTER50

	IF EDGEPOS(in) AND NOT reset THEN
		(* setze Zeitstemperl *)
		ti[iCnt]	:=		clock_ms();
		(* suche vergleichs Zähler *)
		IF iCnt - iNum_Max < 0 THEN
			iCmp	:=	iCnt - iNum_Max + iCnt_Max + 1;
		ELSE
			iCmp	:=	iCnt - iNum_Max;
		END_IF
		(* setze Ausgang *)
		IF 	TIME_TO_DINT(ti[iCmp]) <> 0	AND ti[iCnt] - ti[iCmp] < ti_Max AND iNum_Max <> 0 THEN
			out := 	TRUE;
		ELSE
			out	:=	FALSE;
		END_IF
		(* erhoehe Zähler *)
		IF iCnt >= iCnt_Max	THEN				//erhöhe Zähler
			iCnt			:=	0;
		ELSE
			iCnt			:=	iCnt	+	1;
		END_IF
	ELSIF reset THEN
		(* setze alle variablen zurueck *)
		FOR iCnt := 0 TO iCnt_Max DO
			ti[iCnt]	:=		T#0s;
		END_FOR
		out		:=	FALSE;
		iCnt	:=	0;
		iCmp	:=	0;
	ELSIF out THEN
		IF 	TIME_TO_DINT(ti[iCmp]) <> 0	AND clock_ms() - ti[iCmp] < ti_Max AND iNum_Max <> 0 THEN
			out := 	TRUE;
		ELSE
			out	:=	FALSE;
		END_IF
	END_IF

END_FUNCTION_BLOCK

FUNCTION_BLOCK COUNTER100

	IF EDGEPOS(in) AND NOT reset THEN
		(* setze Zeitstemperl *)
		ti[iCnt]	:=		clock_ms();
		(* suche vergleichs Zähler *)
		IF iCnt - iNum_Max < 0 THEN
			iCmp	:=	iCnt - iNum_Max + iCnt_Max + 1;
		ELSE
			iCmp	:=	iCnt - iNum_Max;
		END_IF
		(* setze Ausgang *)
		IF 	TIME_TO_DINT(ti[iCmp]) <> 0	AND ti[iCnt] - ti[iCmp] < ti_Max AND iNum_Max <> 0 THEN
			out := 	TRUE;
		ELSE
			out	:=	FALSE;
		END_IF
		(* erhoehe Zähler *)
		IF iCnt >= iCnt_Max	THEN				//erhöhe Zähler
			iCnt			:=	0;
		ELSE
			iCnt			:=	iCnt	+	1;
		END_IF
	ELSIF reset THEN
		(* setze alle variablen zurueck *)
		FOR iCnt := 0 TO iCnt_Max DO
			ti[iCnt]	:=		T#0s;
		END_FOR
		out		:=	FALSE;
		iCnt	:=	0;
		iCmp	:=	0;
	ELSIF out THEN
		IF 	TIME_TO_DINT(ti[iCmp]) <> 0	AND clock_ms() - ti[iCmp] < ti_Max AND iNum_Max <> 0 THEN
			out := 	TRUE;
		ELSE
			out	:=	FALSE;
		END_IF
	END_IF

END_FUNCTION_BLOCK
```

#### rmedian.st
```iecst
(********************************************************************
 * COPYRIGHT -- INNIO Company
 ********************************************************************
 * Package: TPSA_lib
 * File: rmedian.st
 * Author: WaldharM
 * Created: March 14, 2012
 *******************************************************************)

FUNCTION_BLOCK RMEDIAN24
	anzahl := LIMIT(0,anzahl,24);
	FOR i := 2 TO anzahl DO
		j := i;
		WHILE j >= 2 AND in[j-1] > in[j] DO
			rDummy := in[j-1];
			in[j-1] := in[j];
			in[j] 	:= rDummy;
			j := j-1;
		END_WHILE
	END_FOR

	IF INT_TO_BOOL(anzahl MOD 2) THEN	// ungerade
		median := in[(anzahl+1)/2];
	ELSE 					//gerade
		median := (in[anzahl/2] + in[anzahl/2+1])/2;
	END_IF
END_FUNCTION_BLOCK
```

#### OP_func.st
```iecst
(********************************************************************

This code is confidential and proprietary to the INNIO Jenbacher Company.
It may not be used in any form, or reproduced in any manner, without the express
written permission of the INNIO Jenbacher Company.
Copyright, INNIO Jenbacher, 2019

Customized modifications: -
------------------------

History:
-------
V4.07.0	29-01-2019	502423184,  new
		19-02-2019	Perktold,	changed Function name acc. to coding guideline
V4.09.0	03-02-2020	Zuschnig,	TOF always active
		12-02-2020	Zuschnig,	included ParaSetupOk plus 2 sec to enable power reductions

Instructions for use:
--------------------

Outstandings: -
------------

*******************************************************************************)

FUNCTION_BLOCK PRed

	IF bEna AND bParaSetupOk_2s THEN
		memcpy(ADR(rP_Set_Max),iAdr_P_Set_Max,4);
		memcpy(ADR(rP_Set_Act),iAdr_P_Set,4);
		memcpy(ADR(iType_Act),iAdr_P_Type,2);

		IF rP_Set_Act > rP_Red	THEN
			rP_Set_Act	:= rP_Red;
			iType_Act	:= iType;
			xTOF.IN		:=	TRUE;
		ELSE
			xTOF.IN		:=	FALSE;
		END_IF

		rP_Set_Max	:=	MIN(rP_Set_Max, rP_Red);

		memcpy(iAdr_P_Set_Max,ADR(rP_Set_Max),4);
		memcpy(iAdr_P_Set,ADR(rP_Set_Act),4);
		memcpy(iAdr_P_Type,ADR(iType_Act),2);
	ELSE
		xTOF.IN	:=	FALSE;
	END_IF

	xTOF.PT	:=	PT;
	xTOF();
	Q	:=	xTOF.Q;

END_FUNCTION_BLOCK
```

### Library Logical/Libraries/lSim6CTR (ANSIC)

#### lSim6CTR.fun
```iecst
FUNCTION_BLOCK Sim6CTR
  VAR_INPUT
    ssMethodType: SINT;
  END_VAR  VAR_INPUT
        CycleTime : REAL := 0.0099999998; (*Proportional Gain*)
  END_VAR
  VAR_INPUT
        Ts_downSampling_speed : REAL := 0.5000000000; (*DownSampling Time for negative Speed Detection*)
  END_VAR
  VAR_INPUT
        u_min_CBP : REAL; (*minimum value for compressor bypass valve*)
  END_VAR
  VAR_INPUT
        rP_drop_limit : REAL := -500.0000000000; (*Load Drop Trigger value*)
  END_VAR
  VAR_INPUT
        rP_el_LockTV : REAL := 1000.0000000000; (*Lock ThrottleValve hysteresies value*)
  END_VAR
  VAR_INPUT
        rP_el_ReleaseTV : REAL := 900.0000000000; (*Release ThrottleValve hysteresies value*)
  END_VAR
  VAR_INPUT
        rN_ok_offset : REAL := 10.0000000000; (*Engine Speed tolerance offset for load drops*)
  END_VAR
  VAR_INPUT
        u_man_TV : REAL := 90.0000000000; (*manual set value for throttle valve*)
  END_VAR
  VAR_INPUT
        u_max_TV : REAL := 1000.0000000000; (*maximum value for throttle valve*)
  END_VAR
  VAR_INPUT
        u_min_TV : REAL; (*minimum value for throttle valve*)
  END_VAR
  VAR_INPUT
        u_max_CBP : REAL := 1000.0000000000; (*maximum value for compressor bypass valve*)
  END_VAR
  VAR_INPUT
        bInit : BOOL := FALSE; (*Init CTR in Tracking Mode*)
  END_VAR
  VAR_INPUT
        Init_Value_CBP : REAL; (*init value compressor bypass*)
  END_VAR
  VAR_INPUT
        w_set : REAL; (*set value*)
  END_VAR
  VAR_INPUT
        x_act : REAL; (*actual value*)
  END_VAR
  VAR_INPUT
        P_CBP : REAL; (*P gain of compressor bypass*)
  END_VAR
  VAR_INPUT
        D_CBP : REAL; (*D gain of compressor bypass*)
  END_VAR
  VAR_OUTPUT
        rPos_CBP : REAL; (*Controller Output*)
  END_VAR
  VAR_INPUT
        rN_act : REAL; (*engine speed actual value*)
  END_VAR
  VAR_INPUT
        rN_set : REAL; (*engine speed set value*)
  END_VAR
  VAR_INPUT
        rP_el : REAL; (*electrical power*)
  END_VAR
  VAR_INPUT
        Init_Value_TV : REAL; (*init value throttle bypass*)
  END_VAR
  VAR_INPUT
        P_TV : REAL; (*P gain of throttle valve*)
  END_VAR
  VAR_INPUT
        D_TV : REAL; (*D gain of throttle valve*)
  END_VAR
  VAR_OUTPUT
        rPos_TV : REAL; (*Controller Output*)
  END_VAR
  VAR_OUTPUT
        rN_act_Diff : REAL; (*test output*)
  END_VAR
  VAR_OUTPUT
        bOpen4CBP : BOOL := FALSE; (*open compressor bypass valve 3 and 4*)
  END_VAR
  VAR_OUTPUT
        bLoadDrop : BOOL := FALSE; (*indication of a load drop*)
  END_VAR
  VAR_OUTPUT
        Control_State : INT; (*indication of a load drop*)
  END_VAR
  VAR_OUTPUT
        bLock_TV : BOOL := FALSE; (*freeze throttle valve to constant value*)
  END_VAR
  VAR_OUTPUT
        bN_ok : BOOL := FALSE; (*test output*)
  END_VAR
  VAR_OUTPUT
        bN_rate_neg : BOOL := FALSE; (*test output*)
  END_VAR
  VAR_OUTPUT
        bP_drop : BOOL := FALSE; (*test output*)
  END_VAR
  VAR_OUTPUT
        rP_grad : REAL; (*test output*)
  END_VAR
  VAR_OUTPUT
        rN_act_DS : REAL; (*test output*)
  END_VAR
  VAR_INPUT
        I_CBP : REAL; (*I gain of compressor bypass*)
  END_VAR
  VAR_INPUT
        I_TV : REAL; (*I gain of throttle valve*)
  END_VAR
	VAR
		bur_Sim6CTR_DWork : D_Work_Sim6CTR;
	END_VAR
	VAR
		bur_Sim6CTR_B : BlockIO_Sim6CTR;
	END_VAR
END_FUNCTION_BLOCK
```

#### lSim6CTR.typ
```iecst
 TYPE

END_TYPE
TYPE
	D_Work_Sim6CTR : STRUCT

		Integrator_DSTATE : REAL;
		Filter_DSTATE : REAL;
		UnitDelay_DSTATE : REAL;
		UnitDelay_DSTATE_e : REAL;
		UD_DSTATE : REAL;
		Delay_DSTATE : ARRAY[0..9] OF REAL;
		UnitDelay_DSTATE_n : REAL;
		Integrator_DSTATE_i : REAL;
		Filter_DSTATE_e : REAL;
		UnitDelay2_DSTATE : BOOL;
		is_active_c1_Sim6CTR : USINT;
		is_c1_Sim6CTR : USINT;
		is_Standard : USINT;
		is_LoadDrop : USINT;
	END_STRUCT;

	 BlockIO_Sim6CTR : STRUCT

		Input11 : REAL;
		Input1 : REAL;
		Input9 : REAL;
		Input3 : REAL;
		Input5 : REAL;
		Modeswitch : REAL;
		Input13 : REAL;
		Input12 : REAL;
		Switch : REAL;
		Diff : REAL;
		Input2 : REAL;
		Add1 : REAL;
		Input14 : REAL;
		Input6 : REAL;
		Input8 : REAL;
		Modeswitch_a : REAL;
		Input4 : REAL;
		Input7 : REAL;
		Control_State : INT;
		Input10 : BOOL;
		RelationalOperator1 : BOOL;
		Compare : BOOL;
		RelationalOperator : BOOL;
		Lock_TV : BOOL;
		bLoadDrop : BOOL;
		Open4CBP : BOOL;
	END_STRUCT;

END_TYPE
```

#### Sim6CTR.h
```c
/********************************************************************
 * COPYRIGHT -- Bernecker + Rainer Industrie-Elektronik Ges.m.b.H.
 ********************************************************************
 * Program: Sim6CTR
 * File: Sim6CTR.h
 * Author: 105051472
 * Created: Wed Oct 23 10:19:46 2013
 ********************************************************************
 * Header for program Sim6CTR
 ********************************************************************
 * Generated with B&R Automation Studio Target for Simulink V4.0
 * (ERT based)
 ********************************************************************/

#ifndef RTW_HEADER_Sim6CTR_h_
#define RTW_HEADER_Sim6CTR_h_
#ifndef Sim6CTR_COMMON_INCLUDES_
# define Sim6CTR_COMMON_INCLUDES_
#include <math.h>
#include "rtwtypes.h"
#endif                                 /* Sim6CTR_COMMON_INCLUDES_ */

#include "Sim6CTR_types.h"
#include "lSim6CTR.h"

/* Macros for accessing real-time model data structure */
#ifndef rtmGetErrorStatus
# define rtmGetErrorStatus(rtm)        ((void*) 0)
#endif

#ifndef rtmSetErrorStatus
# define rtmSetErrorStatus(rtm, val)   ((void) 0)
#endif

#ifndef rtmGetStopRequested
# define rtmGetStopRequested(rtm)      ((void*) 0)
#endif

#ifndef MIN
#define MIN(a,b)                       ((a) < (b) ? (a) : (b))
#endif

#ifndef MAX
#define MAX(a,b)                       ((a) > (b) ? (a) : (b))
#endif

/* Block signals (auto storage) */

/* Block states (auto storage) for system '<Root>' */

/* Block signals (auto storage) */
extern BlockIO_Sim6CTR Sim6CTR_B;

/* Block states (auto storage) */
extern D_Work_Sim6CTR Sim6CTR_DWork;

/* Model entry point functions */
extern void Sim6CTR_initialize(struct Sim6CTR* inst);
extern void Sim6CTR_step(struct Sim6CTR* inst);
extern void Sim6CTR_terminate(struct Sim6CTR* inst);

/*-
 * The generated code includes comments that allow you to trace directly
 * back to the appropriate location in the model.  The basic format
 * is <system>/block_name, where system is the system number (uniquely
 * assigned by Simulink) and block_name is the name of the block.
 *
 * Use the MATLAB hilite_system command to trace the generated code back
 * to the model.  For example,
 *
 * hilite_system('<S3>')    - opens system 3
 * hilite_system('<S3>/Kp') - opens and selects block Kp which resides in S3
 *
 * Here is the system hierarchy for this model
 *
 * '<Root>' : 'Sim6CTR'
 * '<S1>'   : 'Sim6CTR/Island Controller'
 * '<S2>'   : 'Sim6CTR/Model Info'
 * '<S3>'   : 'Sim6CTR/Island Controller/Chart'
 * '<S4>'   : 'Sim6CTR/Island Controller/Compare To Constant1'
 * '<S5>'   : 'Sim6CTR/Island Controller/Difference1'
 * '<S6>'   : 'Sim6CTR/Island Controller/Down Sampling'
 * '<S7>'   : 'Sim6CTR/Island Controller/PID CBP'
 * '<S8>'   : 'Sim6CTR/Island Controller/PID TV'
 * '<S9>'   : 'Sim6CTR/Island Controller/Down Sampling/Timer'
 * '<S10>'  : 'Sim6CTR/Island Controller/PID CBP/PID'
 * '<S11>'  : 'Sim6CTR/Island Controller/PID CBP/PID/Clamping circuit'
 * '<S12>'  : 'Sim6CTR/Island Controller/PID CBP/PID/Clamping circuit/Compare To Constant'
 * '<S13>'  : 'Sim6CTR/Island Controller/PID TV/PID'
 * '<S14>'  : 'Sim6CTR/Island Controller/PID TV/PID/Clamping circuit'
 * '<S15>'  : 'Sim6CTR/Island Controller/PID TV/PID/Clamping circuit/Compare To Constant'
 */
#endif                                 /* RTW_HEADER_Sim6CTR_h_ */
```

#### Sim6CTR_private.h
```c
/********************************************************************
 * COPYRIGHT -- Bernecker + Rainer Industrie-Elektronik Ges.m.b.H.
 ********************************************************************
 * Program: Sim6CTR
 * File: Sim6CTR_private.h
 * Author: 105051472
 * Created: Wed Oct 23 10:19:46 2013
 ********************************************************************
 * Header for program Sim6CTR
 ********************************************************************
 * Generated with B&R Automation Studio Target for Simulink V4.0
 * (ERT based)
 ********************************************************************/

#ifndef RTW_HEADER_Sim6CTR_private_h_
#define RTW_HEADER_Sim6CTR_private_h_
#include "rtwtypes.h"
#include <bur/plctypes.h>
#ifndef __RTWTYPES_H__
#error This file requires rtwtypes.h to be included
#else
#ifdef TMWTYPES_PREVIOUSLY_INCLUDED
#error This file requires rtwtypes.h to be included before tmwtypes.h
#else

/* Check for inclusion of an incorrect version of rtwtypes.h */
#ifndef RTWTYPES_ID_C08S16I32L32N32F1
#error This code was generated with a different "rtwtypes.h" than the file included
#endif                                 /* RTWTYPES_ID_C08S16I32L32N32F1 */
#endif                                 /* TMWTYPES_PREVIOUSLY_INCLUDED */
#endif                                 /* __RTWTYPES_H__ */

#ifndef MIN
#define MIN(a,b)                       ((a) < (b) ? (a) : (b))
#endif

#ifndef MAX
#define MAX(a,b)                       ((a) > (b) ? (a) : (b))
#endif

/* Imported (extern) block parameters */
extern real32_T CycleTime;             /* Variable: CycleTime
                                        * Referenced by: '<S1>/Cyclic Time'
                                        */
extern real32_T Ts_downSampling_speed; /* Variable: Ts_downSampling_speed
                                        * Referenced by: '<S1>/Ts_downSampling_speed'
                                        */
extern real32_T rN_ok_offset;          /* Variable: rN_ok_offset
                                        * Referenced by: '<S1>/rN_ok_offset'
                                        */
extern real32_T rP_drop_limit;         /* Variable: rP_drop_limit
                                        * Referenced by: '<S1>/rP_drop_limit'
                                        */
extern real32_T rP_el_LockTV;          /* Variable: rP_el_LockTV
                                        * Referenced by: '<S1>/rP_el_LockTV'
                                        */
extern real32_T rP_el_ReleaseTV;       /* Variable: rP_el_ReleaseTV
                                        * Referenced by: '<S1>/rP_el_ReleaseTV'
                                        */
extern real32_T u_man_TV;              /* Variable: u_man_TV
                                        * Referenced by: '<S1>/u_man_TV'
                                        */
extern real32_T u_max_CBP;             /* Variable: u_max_CBP
                                        * Referenced by: '<S10>/Saturation'
                                        */
extern real32_T u_max_TV;              /* Variable: u_max_TV
                                        * Referenced by: '<S13>/Saturation'
                                        */
extern real32_T u_min_CBP;             /* Variable: u_min_CBP
                                        * Referenced by: '<S10>/Saturation'
                                        */
extern real32_T u_min_TV;              /* Variable: u_min_TV
                                        * Referenced by: '<S13>/Saturation'
                                        */

#endif                                 /* RTW_HEADER_Sim6CTR_private_h_ */
```

#### Sim6CTR_types.h
```c
/********************************************************************
 * COPYRIGHT -- Bernecker + Rainer Industrie-Elektronik Ges.m.b.H.
 ********************************************************************
 * Program: Sim6CTR
 * File: Sim6CTR_types.h
 * Author: 105051472
 * Created: Wed Oct 23 10:19:46 2013
 ********************************************************************
 * Header for program Sim6CTR
 ********************************************************************
 * Generated with B&R Automation Studio Target for Simulink V4.0
 * (ERT based)
 ********************************************************************/

#ifndef RTW_HEADER_Sim6CTR_types_h_
#define RTW_HEADER_Sim6CTR_types_h_
#ifndef MIN
#define MIN(a,b)                       ((a) < (b) ? (a) : (b))
#endif

#ifndef MAX
#define MAX(a,b)                       ((a) > (b) ? (a) : (b))
#endif
#endif                                 /* RTW_HEADER_Sim6CTR_types_h_ */
```

#### rtwtypes.h
```c
/********************************************************************
 * COPYRIGHT -- Bernecker + Rainer Industrie-Elektronik Ges.m.b.H.
 ********************************************************************
 * Program: Sim6CTR
 * File: rtwtypes.h
 * Author: 105051472
 * Created: Wed Oct 23 10:19:46 2013
 ********************************************************************
 * Header for program Sim6CTR
 ********************************************************************
 * Generated with B&R Automation Studio Target for Simulink V4.0
 * (ERT based)
 ********************************************************************/

#ifndef __RTWTYPES_H__
#define __RTWTYPES_H__
#ifndef TRUE
# define TRUE                          (1U)
#endif

#ifndef FALSE
# define FALSE                         (0U)
#endif

#ifndef __TMWTYPES__
#define __TMWTYPES__
#include <limits.h>

/*=======================================================================*
 * Target hardware information
 *   Device type: Intel->x86/Pentium
 *   Number of bits:     char:   8    short:   16    int:  32
 *                       long:  32
 *                       native word size:  32
 *   Byte ordering: LittleEndian
 *   Signed integer division rounds to: Zero
 *   Shift right on a signed integer as arithmetic shift: on
 *=======================================================================*/

/*=======================================================================*
 * Fixed width word size data types:                                     *
 *   int8_T, int16_T, int32_T     - signed 8, 16, or 32 bit integers     *
 *   uint8_T, uint16_T, uint32_T  - unsigned 8, 16, or 32 bit integers   *
 *   real32_T, real64_T           - 32 and 64 bit floating point numbers *
 *=======================================================================*/
typedef signed char int8_T;
typedef unsigned char uint8_T;
typedef short int16_T;
typedef unsigned short uint16_T;
typedef int int32_T;
typedef unsigned int uint32_T;
typedef float real32_T;
typedef double real64_T;

/*===========================================================================*
 * Generic type definitions: real_T, time_T, boolean_T, int_T, uint_T,       *
 *                           ulong_T, char_T and byte_T.                     *
 *===========================================================================*/
typedef double real_T;
typedef double time_T;
typedef unsigned char boolean_T;
typedef int int_T;
typedef unsigned int uint_T;
typedef unsigned long ulong_T;
typedef char char_T;
typedef unsigned char uchar_T;
typedef char_T byte_T;

/*=======================================================================*
 * Min and Max:                                                          *
 *   int8_T, int16_T, int32_T     - signed 8, 16, or 32 bit integers     *
 *   uint8_T, uint16_T, uint32_T  - unsigned 8, 16, or 32 bit integers   *
 *=======================================================================*/
#define MAX_int8_T                     ((int8_T)(127))
#define MIN_int8_T                     ((int8_T)(-128))
#define MAX_uint8_T                    ((uint8_T)(255U))
#define MIN_uint8_T                    ((uint8_T)(0U))
#define MAX_int16_T                    ((int16_T)(32767))
#define MIN_int16_T                    ((int16_T)(-32768))
#define MAX_uint16_T                   ((uint16_T)(65535U))
#define MIN_uint16_T                   ((uint16_T)(0U))
#define MAX_int32_T                    ((int32_T)(2147483647))
#define MIN_int32_T                    ((int32_T)(-2147483647-1))
#define MAX_uint32_T                   ((uint32_T)(0xFFFFFFFFU))
#define MIN_uint32_T                   ((uint32_T)(0U))

/* Logical type definitions */
#if (!defined(__cplusplus)) && (!defined(__true_false_are_keywords))
#  ifndef false
#   define false                       (0U)
#  endif

#  ifndef true
#   define true                        (1U)
#  endif
#endif

/*
 * Simulink Coder assumes the code is compiled on a target using a 2's complement representation
 * for signed integer values.
 */
#if ((SCHAR_MIN + 1) != -SCHAR_MAX)
#error "This code must be compiled using a 2's complement representation for signed integer values"
#endif

/* This ID is used to detect inclusion of an incompatible rtwtypes.h */
#define RTWTYPES_ID_C08S16I32L32N32F1
#else                                  /* __TMWTYPES__ */
#define TMWTYPES_PREVIOUSLY_INCLUDED
#endif                                 /* __TMWTYPES__ */

/* Block D-Work pointer type */
typedef void * pointer_T;

/* Simulink specific types */
#ifndef __SIMSTRUC_TYPES_H__
#define __SIMSTRUC_TYPES_H__

/* Trigger directions: falling, either, and rising */
typedef enum {
  FALLING_ZERO_CROSSING = -1,
  ANY_ZERO_CROSSING = 0,
  RISING_ZERO_CROSSING = 1
} ZCDirection;

/* Previous state of a trigger signal */
typedef uint8_T ZCSigState;

/* Initial value of a trigger zero crossing signal */
#define UNINITIALIZED_ZCSIG            0x03U
#define NEG_ZCSIG                      0x02U
#define POS_ZCSIG                      0x01U
#define ZERO_ZCSIG                     0x00U

/* Current state of a trigger signal */
typedef enum {
  FALLING_ZCEVENT = -1,
  NO_ZCEVENT = 0,
  RISING_ZCEVENT = 1
} ZCEventType;

#endif                                 /* __SIMSTRUC_TYPES_H__ */
#endif                                 /* __RTWTYPES_H__ */

#ifndef MIN
#define MIN(a,b)                       ((a) < (b) ? (a) : (b))
#endif

#ifndef MAX
#define MAX(a,b)                       ((a) > (b) ? (a) : (b))
#endif
```
